RoboDK station: FranciscoPantoja_Tarea4_seguimiento.rdk

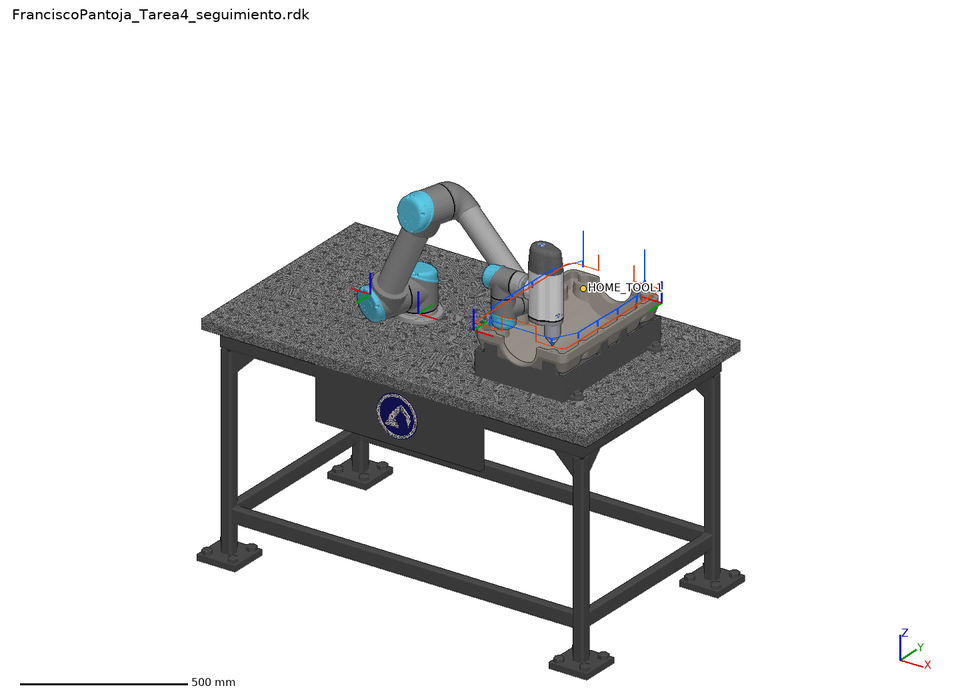
[picture v0: the station drawn from its stored meshes, robots at their saved joint values, targets as dots, program paths as lines]
Station Block1 (saved by RoboDK 5.5.1). Poses are relative to the parent item; angles as X-Y-Z fixed-axis rotations.
Station parameters (name, value as stored): ViewNames, New View 1|[19.806,-223.251,-1852.955,-4.394,-26.413,-81.026]||New View 2|[-145.353,-147.123,-1133.187,-12.666,-29.479,-64.252]||New View 3|[-89.962,-117.618,-1053.622,-35.524,-65.339,-53.555]||New View 4|[104.763,80.763,-3406.264,-32.675,-38.414,-42.423]||, TAGS, ['Dispensing'], Palletizing Plugin
  - frame World at (0, 0, 0) mm
    - object Table at (0, 0, 0) mm, size 1420 x 820 x 800 mm, geometry from Table-1400x800x800.sld
    - frame Doosan Robotics M1013 - Navy Base at (-392.37, 24.39, 0) mm, rotated rx 0 ry 0 rz -180 deg
      - frame Part at (-900, -230, 130) mm
        - object Pan_Holder at (0, 0, 0) mm, size 400 x 503 x 157.6 mm, geometry from Jig2.step
        - object Part_Oil_Pan at (0, 0, 0) mm, size 330.2 x 509.8 x 126.9 mm, 15 curves
    - target HOME_TOOL1 (Cartesian target) at (400, 0, 250) mm, rotated rx -180 ry 0 rz 180 deg; joints [15.487, -80.374, -104.044, -47.614, 80.326, 102.152] of UR5
  - frame UR5 Base at (-200, 0, 0) mm
    - robot UR5: 6 axes
        modified DH rows (alpha deg, a mm, theta deg, d mm): 0, 0, 0, 89.2; 90, 0, 180, 0; 0, 425, 0, 0; 0, 392, 0, 109.3; -90, 0, 0, 94.75; 90, 0, 0, 82.5
        joint limits [-360, -360, -360, -360, -360, -360] to [360, 360, 360, 360, 360, 360]; home [0, -90, -90, 0, 90, 0]; saved at [-15.092, -117.834, -95.599, 33.433, 105.092, 90]
      - tool OnRobot Screwdriver, TCP at (168.4, 0, 95.37) mm, rotated rx 0 ry 90 rz 0 deg, size 323.9 x 86.2 x 125.3 mm
      - tool Spintech Spindle, TCP at (32, 0, 260) mm, rotated rx 0 ry 39 rz 0 deg, size 157.3 x 72 x 259.9 mm
  - machining project Path1 ajustes: rotZ(0) | rotX(0)*rotY(0) | rotz(0) | onStart | onPathStart | onApproach | onPoint | onRetract | onFinish | SetRPM(%1) | SetTool(%1) | Extruder(%1) | default | default | OutOnMov(%1) | OutOffMov(%1) | onPathFinish | M_RunCode(%1)
  - machining project Ajustes de puntos: rotZ(0) | rotX(0)*rotY(0) | onStart | onPathStart | onApproach | onPoint | onRetract | onFinish | SetRPM(%1) | SetTool(%1) | Extruder(%1) | default | default | OutOnMov(%1) | OutOffMov(%1) | onPathFinish | M_RunCode(%1)
  - program Ajustes (71 instructions, listed below)
  - program Path1 (47 instructions, listed below)
  - program MAIN (7 instructions, listed below)
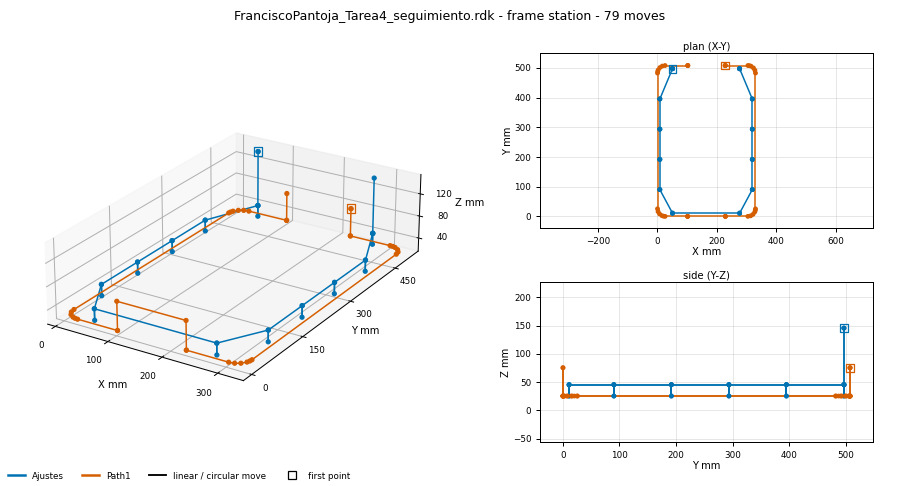
[picture p0: tool path of FranciscoPantoja_Tarea4_seguimiento.rdk in frame station, 79 of 79 moves have a stored position in this frame; points joined in program order, loops and branches not executed]

--- program Ajustes (robot UR5) ---
  Suave(1)
  Establecer velocidad (1000.0 mm/s)
  Est. Ref.: World
  Est. herr: OnRobot Screwdriver
  Mostrar OnRobot Screwdriver
  MoveJ 1 to (50.77, 496.76, 145.4) mm, rotated rx -180 ry 0 rz 0 deg; joints [-15.092, -111.753, -88.373, 20.126, 105.092, 90]
  MoveL 2 to (50.77, 496.76, 145.4) mm, rotated rx -180 ry 0 rz 0 deg; joints [-15.092, -111.753, -88.373, 20.126, 105.092, 90]
  MoveL 3 to (50.77, 496.76, 45.4) mm, rotated rx -180 ry 0 rz 0 deg; joints [-15.092, -117.834, -95.599, 33.433, 105.092, 90]
  MoveL 4 to (50.77, 496.76, 45.4) mm, rotated rx -180 ry 0 rz 0 deg; joints [-15.092, -117.834, -95.599, 33.433, 105.092, 90]
  Establecer velocidad (30.0 mm/s)
  MoveL 5 to (50.77, 496.76, 25.4) mm, rotated rx -180 ry 0 rz 0 deg; joints [-15.092, -119.379, -96.636, 36.015, 105.092, 90]
  MoveL 6 to (50.77, 496.76, 45.4) mm, rotated rx -180 ry 0 rz 0 deg; joints [-15.092, -117.834, -95.599, 33.433, 105.092, 90]
  Establecer velocidad (1000.0 mm/s)
  MoveL 7 to (8.24, 395.16, 45.4) mm, rotated rx -180 ry 0 rz 0 deg; joints [-3.432, -118.223, -94.973, 33.196, 93.432, 90]
  Establecer velocidad (30.0 mm/s)
  MoveL 8 to (8.24, 395.16, 25.4) mm, rotated rx -180 ry 0 rz 0 deg; joints [-3.432, -119.757, -96.009, 35.765, 93.432, 90]
  MoveL 9 to (8.24, 395.16, 45.4) mm, rotated rx -180 ry 0 rz 0 deg; joints [-3.432, -118.223, -94.973, 33.196, 93.432, 90]
  Establecer velocidad (1000.0 mm/s)
  MoveL 10 to (8.24, 293.56, 45.4) mm, rotated rx -180 ry 0 rz 0 deg; joints [7.768, -116.241, -98.138, 34.379, 82.232, 90]
  Establecer velocidad (30.0 mm/s)
  MoveL 11 to (8.24, 293.56, 25.4) mm, rotated rx -180 ry 0 rz 0 deg; joints [7.768, -117.833, -99.181, 37.013, 82.232, 90]
  MoveL 12 to (8.24, 293.56, 45.4) mm, rotated rx -180 ry 0 rz 0 deg; joints [7.768, -116.241, -98.138, 34.379, 82.232, 90]
  Establecer velocidad (1000.0 mm/s)
  MoveL 13 to (8.24, 191.96, 45.4) mm, rotated rx -180 ry 0 rz 0 deg; joints [18.837, -116.5, -97.728, 34.228, 71.163, 90]
  Establecer velocidad (30.0 mm/s)
  MoveL 14 to (8.24, 191.96, 25.4) mm, rotated rx -180 ry 0 rz 0 deg; joints [18.837, -118.084, -98.769, 36.853, 71.163, 90]
  MoveL 15 to (8.24, 191.96, 45.4) mm, rotated rx -180 ry 0 rz 0 deg; joints [18.837, -116.5, -97.728, 34.228, 71.163, 90]
  Establecer velocidad (1000.0 mm/s)
  MoveL 16 to (8.24, 90.36, 45.4) mm, rotated rx -180 ry 0 rz 0 deg; joints [28.992, -118.978, -93.75, 32.729, 61.008, 90]
  Establecer velocidad (30.0 mm/s)
  MoveL 17 to (8.24, 90.36, 25.4) mm, rotated rx -180 ry 0 rz 0 deg; joints [28.992, -120.491, -94.784, 35.275, 61.008, 90]
  MoveL 18 to (8.24, 90.36, 45.4) mm, rotated rx -180 ry 0 rz 0 deg; joints [28.992, -118.978, -93.75, 32.729, 61.008, 90]
  Establecer velocidad (1000.0 mm/s)
  MoveL 19 to (50.77, 11.24, 45.4) mm, rotated rx -180 ry 0 rz 0 deg; joints [38.653, -117.875, -95.534, 33.409, 51.347, 90]
  Establecer velocidad (30.0 mm/s)
  MoveL 20 to (50.77, 11.24, 25.4) mm, rotated rx -180 ry 0 rz 0 deg; joints [38.653, -119.418, -96.571, 35.989, 51.347, 90]
  MoveL 21 to (50.77, 11.24, 45.4) mm, rotated rx -180 ry 0 rz 0 deg; joints [38.653, -117.875, -95.534, 33.409, 51.347, 90]
  Establecer velocidad (1000.0 mm/s)
  MoveL 22 to (276.5, 11.24, 45.4) mm, rotated rx -180 ry 0 rz 0 deg; joints [61.971, -95.798, -126.335, 42.133, 28.029, 90]
  Establecer velocidad (30.0 mm/s)
  MoveL 23 to (276.5, 11.24, 25.4) mm, rotated rx 180 ry 0 rz 0 deg; joints [61.971, -98.141, -127.625, 45.766, 28.029, 90]
  MoveL 24 to (276.5, 11.24, 45.4) mm, rotated rx -180 ry 0 rz 0 deg; joints [61.971, -95.798, -126.335, 42.133, 28.029, 90]
  Establecer velocidad (1000.0 mm/s)
  MoveL 25 to (319.03, 90.36, 45.4) mm, rotated rx -180 ry 0 rz 0 deg; joints [62.057, -83.585, -138.453, 42.037, 27.943, 90]
  Establecer velocidad (30.0 mm/s)
  MoveL 26 to (319.03, 90.36, 25.4) mm, rotated rx 180 ry 0 rz 0 deg; joints [62.057, -86.468, -140.031, 46.499, 27.943, 90]
  MoveL 27 to (319.03, 90.36, 45.4) mm, rotated rx -180 ry 0 rz 0 deg; joints [62.057, -83.585, -138.453, 42.037, 27.943, 90]
  Establecer velocidad (1000.0 mm/s)
  MoveL 28 to (319.03, 191.96, 45.4) mm, rotated rx 180 ry 0 rz 0 deg; joints [46.324, -74.874, -144.831, 39.706, 43.676, 90]
  Establecer velocidad (30.0 mm/s)
  MoveL 29 to (319.03, 191.96, 25.4) mm, rotated rx -180 ry 0 rz 0 deg; joints [46.324, -78.094, -146.663, 44.757, 43.676, 90]
  MoveL 30 to (319.03, 191.96, 45.4) mm, rotated rx 180 ry 0 rz 0 deg; joints [46.324, -74.874, -144.831, 39.706, 43.676, 90]
  Establecer velocidad (1000.0 mm/s)
  MoveL 31 to (319.03, 293.56, 45.4) mm, rotated rx -180 ry 0 rz 0 deg; joints [20.13, -73.726, -145.543, 39.269, 69.87, 90]
  Establecer velocidad (30.0 mm/s)
  MoveL 32 to (319.03, 293.56, 25.4) mm, rotated rx -180 ry 0 rz 0 deg; joints [20.13, -76.982, -147.409, 44.392, 69.87, 90]
  MoveL 33 to (319.03, 293.56, 45.4) mm, rotated rx -180 ry 0 rz 0 deg; joints [20.13, -73.726, -145.543, 39.269, 69.87, 90]
  Establecer velocidad (1000.0 mm/s)
  MoveL 34 to (319.03, 395.16, 45.4) mm, rotated rx -180 ry 0 rz 0 deg; joints [-8.193, -81.267, -140.326, 41.593, 98.193, 90]
  Establecer velocidad (30.0 mm/s)
  MoveL 35 to (319.03, 395.16, 25.4) mm, rotated rx -180 ry 0 rz 0 deg; joints [-8.193, -84.248, -141.969, 46.217, 98.193, 90]
  MoveL 36 to (319.03, 395.16, 45.4) mm, rotated rx -180 ry 0 rz 0 deg; joints [-8.193, -81.267, -140.326, 41.593, 98.193, 90]
  Establecer velocidad (1000.0 mm/s)
  MoveL 37 to (276.5, 496.76, 45.4) mm, rotated rx -180 ry 0 rz 0 deg; joints [-25.573, -95.728, -126.415, 42.143, 115.573, 90]
  Establecer velocidad (30.0 mm/s)
  MoveL 38 to (276.5, 496.76, 25.4) mm, rotated rx 180 ry 0 rz 0 deg; joints [-25.573, -98.074, -127.707, 45.781, 115.573, 90]
  MoveL 39 to (276.5, 496.76, 45.4) mm, rotated rx -180 ry 0 rz 0 deg; joints [-25.573, -95.728, -126.415, 42.143, 115.573, 90]
  MoveL 40 to (276.5, 496.76, 45.4) mm, rotated rx -180 ry 0 rz 0 deg; joints [-25.573, -95.728, -126.415, 42.143, 115.573, 90]
  Establecer velocidad (1000.0 mm/s)
  MoveL 41 to (276.5, 496.76, 45.4) mm, rotated rx -180 ry 0 rz 0 deg; joints [-25.573, -95.728, -126.415, 42.143, 115.573, 90]
  MoveL 42 to (276.5, 496.76, 145.4) mm, rotated rx -180 ry 0 rz 0 deg; joints [-25.573, -86.936, -117.883, 24.819, 115.573, 90]

--- program Path1 (robot UR5) ---
  Suave(1)
  Establecer velocidad (1000.0 mm/s)
  Est. Ref.: World
  Est. herr: Spintech Spindle
  Mostrar Spintech Spindle
  MoveJ 1 to (227.98, 507.56, 75.4) mm, rotated rx -180 ry 0 rz 0 deg; joints [-24.692, -77.216, -112.789, -43.651, 105.242, 70.337]
  MoveL 2 to (227.98, 507.56, 75.4) mm, rotated rx -180 ry 0 rz 0 deg; joints [-24.692, -77.216, -112.789, -43.651, 105.242, 70.337]
  MoveL 3 to (227.98, 507.56, 25.4) mm, rotated rx -180 ry 0 rz 0 deg; joints [-24.692, -79.026, -118.933, -35.697, 105.242, 70.337]
  MoveL 4 to (227.98, 507.56, 25.4) mm, rotated rx -180 ry 0 rz 0 deg; joints [-24.692, -79.026, -118.933, -35.697, 105.242, 70.337]
  Establecer velocidad (50.0 mm/s)
  MoveL 5 to (304.36, 507.56, 25.4) mm, rotated rx -180 ry 0 rz 0 deg; joints [-30.672, -70.135, -124.849, -40.159, 108.725, 65.254]
  MoveL 6 to (309.56, 507.02, 25.4) mm, rotated rx 180 ry 0 rz 0 deg; joints [-31.08, -69.481, -125.226, -40.55, 108.958, 64.9]
  MoveL 7 to (314.85, 505.29, 25.4) mm, rotated rx -180 ry 0 rz 0 deg; joints [-31.316, -68.671, -125.699, -40.954, 109.093, 64.695]
  MoveL 8 to (322.91, 499.51, 25.4) mm, rotated rx -180 ry 0 rz 0 deg; joints [-31.17, -67.032, -126.656, -41.595, 109.009, 64.822]
  MoveL 9 to (327.94, 491.61, 25.4) mm, rotated rx -180 ry 0 rz 0 deg; joints [-30.329, -65.442, -127.58, -42.027, 108.529, 65.55]
  MoveL 10 to (329.76, 482.16, 25.4) mm, rotated rx -180 ry 0 rz 0 deg; joints [-28.824, -64.004, -128.417, -42.225, 107.662, 66.846]
  MoveL 11 to (329.76, 25.84, 25.4) mm, rotated rx -180 ry 0 rz 0 deg; joints [72.393, -60.789, -125.212, -70.235, 53.142, 157.787]
  MoveL 12 to (329.22, 20.64, 25.4) mm, rotated rx -180 ry 0 rz 0 deg; joints [72.61, -61.544, -124.817, -70.034, 53.09, 158.051]
  MoveL 13 to (327.49, 15.35, 25.4) mm, rotated rx 180 ry 0 rz 0 deg; joints [72.596, -62.455, -124.375, -69.555, 53.093, 158.034]
  MoveL 14 to (321.71, 7.29, 25.4) mm, rotated rx 180 ry 0 rz 0 deg; joints [71.993, -64.204, -123.588, -68.154, 53.238, 157.302]
  MoveL 15 to (313.81, 2.26, 25.4) mm, rotated rx 180 ry 0 rz 0 deg; joints [70.868, -65.792, -122.927, -66.417, 53.519, 155.945]
  MoveL 16 to (304.36, 0.44, 25.4) mm, rotated rx 180 ry 0 rz 0 deg; joints [69.335, -67.153, -122.418, -64.479, 53.926, 154.111]
  MoveL 17 to (228.6, 0.44, 25.4) mm, rotated rx 180 ry 0 rz 0 deg; joints [57.895, -76.655, -117.894, -52.166, 57.786, 141.085]
  Establecer velocidad (1000.0 mm/s)
  MoveL 18 to (228.6, 0.44, 25.4) mm, rotated rx 180 ry 0 rz 0 deg; joints [57.895, -76.655, -117.894, -52.166, 57.786, 141.085]
  MoveL 19 to (228.6, 0.44, 75.4) mm, rotated rx 180 ry 0 rz 0 deg; joints [57.895, -75.284, -111.455, -59.974, 57.786, 141.085]
  Establecer velocidad (1000.0 mm/s)
  MoveL 20 to (101.6, 0.44, 75.4) mm, rotated rx -180 ry 0 rz 0 deg; joints [44.415, -90.899, -99.369, -49.686, 63.869, 127.287]
  MoveL 21 to (101.6, 0.44, 25.4) mm, rotated rx 180 ry 0 rz 0 deg; joints [44.415, -92.569, -105.18, -42.205, 63.869, 127.287]
  MoveL 22 to (101.6, 0.44, 25.4) mm, rotated rx 180 ry 0 rz 0 deg; joints [44.415, -92.569, -105.18, -42.205, 63.869, 127.287]
  Establecer velocidad (50.0 mm/s)
  MoveL 23 to (25.84, 0.44, 25.4) mm, rotated rx 180 ry 0 rz 0 deg; joints [38.744, -101.791, -95.134, -40.799, 66.805, 121.947]
  MoveL 24 to (20.64, 0.98, 25.4) mm, rotated rx -180 ry 0 rz 0 deg; joints [38.359, -102.393, -94.419, -40.773, 67.012, 121.593]
  MoveL 25 to (15.35, 2.71, 25.4) mm, rotated rx 180 ry 0 rz 0 deg; joints [37.875, -102.942, -93.77, -40.701, 67.271, 121.151]
  MoveL 26 to (7.29, 8.49, 25.4) mm, rotated rx 180 ry 0 rz 0 deg; joints [36.892, -103.617, -92.992, -40.462, 67.803, 120.257]
  MoveL 27 to (2.26, 16.39, 25.4) mm, rotated rx -180 ry 0 rz 0 deg; joints [35.929, -103.826, -92.795, -40.125, 68.329, 119.386]
  MoveL 28 to (0.44, 25.84, 25.4) mm, rotated rx -180 ry 0 rz 0 deg; joints [35.026, -103.583, -93.167, -39.702, 68.826, 118.577]
  MoveL 29 to (0.44, 482.16, 25.4) mm, rotated rx -180 ry 0 rz 0 deg; joints [-12.632, -104.392, -93.111, -34.182, 97.911, 80.12]
  MoveL 30 to (0.98, 487.36, 25.4) mm, rotated rx -180 ry 0 rz 0 deg; joints [-13.168, -104.594, -92.839, -34.311, 98.243, 79.695]
  MoveL 31 to (2.71, 492.65, 25.4) mm, rotated rx -180 ry 0 rz 0 deg; joints [-13.74, -104.664, -92.736, -34.411, 98.596, 79.241]
  MoveL 32 to (8.49, 500.71, 25.4) mm, rotated rx -180 ry 0 rz 0 deg; joints [-14.693, -104.41, -93.039, -34.479, 99.185, 78.482]
  MoveL 33 to (16.39, 505.74, 25.4) mm, rotated rx -180 ry 0 rz 0 deg; joints [-15.41, -103.754, -93.858, -34.41, 99.627, 77.91]
  MoveL 34 to (25.84, 507.56, 25.4) mm, rotated rx 180 ry 0 rz 0 deg; joints [-15.862, -102.746, -95.117, -34.22, 99.904, 77.548]
  MoveL 35 to (102.22, 507.56, 25.4) mm, rotated rx -180 ry 0 rz 0 deg; joints [-18.402, -93.812, -105.445, -33.206, 101.459, 75.504]
  Establecer velocidad (1000.0 mm/s)
  MoveL 36 to (102.22, 507.56, 25.4) mm, rotated rx -180 ry 0 rz 0 deg; joints [-18.402, -93.812, -105.445, -33.206, 101.459, 75.504]
  MoveL 37 to (102.22, 507.56, 75.4) mm, rotated rx -180 ry 0 rz 0 deg; joints [-18.402, -91.964, -99.807, -40.691, 101.459, 75.504]

--- program MAIN (robot UR5) ---
  Mostrar Spintech Spindle
  Ocultar OnRobot Screwdriver
  Llamar Path1
  Pausa 2.0 s
  Ocultar Spintech Spindle
  Mostrar OnRobot Screwdriver
  Llamar Ajustes
